Staubli VAL3: designr0.pjx

--- designr0.pjx ---
Parameters version=s7.6.2 stackSize=5000 millimeterUnit=true
Program file=start.pgx
Program file=stop.pgx
Data file=designr0.dtx

--- designr0.dtx ---
mdesc mNomSpeed
pointRx pikk[6 6]
  [0,0] = {x=-175.775864, y=339.495741, z=-126.071808, rx=0.004243, ry=-179.997236, rz=44.99886, fatherId=world[0]}
  [0,1] = {x=-182.38, y=339.495741, z=-126.071808, rx=0.004243, ry=-179.997236, rz=44.99886, fatherId=world[0]}
  [0,2] = {x=-188.98, y=339.5, z=-126, rx=180, ry=0, rz=-135, fatherId=world[0]}
  [0,3] = {x=-195.58, y=339.5, z=-126, rx=180, ry=0, rz=-135, fatherId=world[0]}
  [0,4] = {x=-202.18, y=339.5, z=-126, rx=180, ry=0, rz=-135, fatherId=world[0]}
  [0,5] = {x=-208.78, y=339.5, z=-126, rx=180, ry=0, rz=-135, fatherId=world[0]}
  [1,0] = {x=-175.78, y=349.8, z=-126, rx=180, ry=0, rz=-135, fatherId=world[0]}
  [1,1] = {x=-182.38, y=349.8, z=-126, rx=180, ry=0, rz=-135, fatherId=world[0]}
  [1,2] = {x=-188.98, y=349.8, z=-126, rx=180, ry=0, rz=-135, fatherId=world[0]}
  [1,3] = {x=-195.58, y=349.8, z=-126, rx=180, ry=0, rz=-135, fatherId=world[0]}
  [1,4] = {x=-202.18, y=349.8, z=-126, rx=180, ry=0, rz=-135, fatherId=world[0]}
  [1,5] = {x=-208.78, y=349.8, z=-126, rx=180, ry=0, rz=-135, fatherId=world[0]}
  [2,0] = {x=-175.78, y=360.1, z=-126, rx=180, ry=0, rz=-135, fatherId=world[0]}
  [2,1] = {x=-182.38, y=360.1, z=-126, rx=180, ry=0, rz=-135, fatherId=world[0]}
  [2,2] = {x=-188.98, y=360.1, z=-126, rx=180, ry=0, rz=-135, fatherId=world[0]}
  [2,3] = {x=-195.58, y=360.1, z=-126, rx=180, ry=0, rz=-135, fatherId=world[0]}
  [2,4] = {x=-202.18, y=360.1, z=-126, rx=180, ry=0, rz=-135, fatherId=world[0]}
  [2,5] = {x=-208.78, y=360.1, z=-126, rx=180, ry=0, rz=-135, fatherId=world[0]}
  [3,0] = {x=-175.78, y=370.4, z=-126, rx=180, ry=0, rz=-135, fatherId=world[0]}
  [3,1] = {x=-182.38, y=370.4, z=-126, rx=180, ry=0, rz=-135, fatherId=world[0]}
  [3,2] = {x=-188.98, y=370.4, z=-126, rx=180, ry=0, rz=-135, fatherId=world[0]}
  [3,3] = {x=-195.58, y=370.4, z=-126, rx=180, ry=0, rz=-135, fatherId=world[0]}
  [3,4] = {x=-202.18, y=370.4, z=-126, rx=180, ry=0, rz=-135, fatherId=world[0]}
  [3,5] = {x=-208.78, y=370.4, z=-126, rx=180, ry=0, rz=-135, fatherId=world[0]}
  [4,0] = {x=-175.78, y=380.7, z=-126, rx=180, ry=0, rz=-135, fatherId=world[0]}
  [4,1] = {x=-182.38, y=380.7, z=-126, rx=180, ry=0, rz=-135, fatherId=world[0]}
  [4,2] = {x=-188.98, y=380.7, z=-126, rx=180, ry=0, rz=-135, fatherId=world[0]}
  [4,3] = {x=-195.58, y=380.7, z=-126, rx=180, ry=0, rz=-135, fatherId=world[0]}
  [4,4] = {x=-202.18, y=380.7, z=-126, rx=180, ry=0, rz=-135, fatherId=world[0]}
  [4,5] = {x=-208.78, y=380.7, z=-126, rx=180, ry=0, rz=-135, fatherId=world[0]}
  [5,0] = {x=-175.78, y=391, z=-126, rx=180, ry=0, rz=-135, fatherId=world[0]}
  [5,1] = {x=-182.38, y=391, z=-126, rx=180, ry=0, rz=-135, fatherId=world[0]}
  [5,2] = {x=-188.98, y=391, z=-126, rx=180, ry=0, rz=-135, fatherId=world[0]}
  [5,3] = {x=-195.58, y=391, z=-126, rx=180, ry=0, rz=-135, fatherId=world[0]}
  [5,4] = {x=-202.18, y=391, z=-126, rx=180, ry=0, rz=-135, fatherId=world[0]}
  [5,5] = {x=-208.78, y=391, z=-126.071808, rx=0.004243, ry=-179.997236, rz=44.99886, fatherId=world[0]}
tool pick[6 6]
  [0,0] = {fatherId=flange[0], ioLink=valve1}
  [0,1] = {fatherId=flange[0], ioLink=valve1}
  [0,2] = {fatherId=flange[0], ioLink=valve1}
  [0,3] = {fatherId=flange[0], ioLink=valve1}
  [0,4] = {fatherId=flange[0], ioLink=valve1}
  [0,5] = {fatherId=flange[0], ioLink=valve1}
  [1,0] = {fatherId=flange[0], ioLink=valve1}
  [1,1] = {fatherId=flange[0], ioLink=valve1}
  [1,2] = {fatherId=flange[0], ioLink=valve1}
  [1,3] = {fatherId=flange[0], ioLink=valve1}
  [1,4] = {fatherId=flange[0], ioLink=valve1}
  [1,5] = {fatherId=flange[0], ioLink=valve1}
  [2,0] = {fatherId=flange[0], ioLink=valve1}
  [2,1] = {fatherId=flange[0], ioLink=valve1}
  [2,2] = {fatherId=flange[0], ioLink=valve1}
  [2,3] = {fatherId=flange[0], ioLink=valve1}
  [2,4] = {fatherId=flange[0], ioLink=valve1}
  [2,5] = {fatherId=flange[0], ioLink=valve1}
  [3,0] = {fatherId=flange[0], ioLink=valve1}
  [3,1] = {fatherId=flange[0], ioLink=valve1}
  [3,2] = {fatherId=flange[0], ioLink=valve1}
  [3,3] = {fatherId=flange[0], ioLink=valve1}
  [3,4] = {fatherId=flange[0], ioLink=valve1}
  [3,5] = {fatherId=flange[0], ioLink=valve1}
  [4,0] = {fatherId=flange[0], ioLink=valve1}
  [4,1] = {fatherId=flange[0], ioLink=valve1}
  [4,2] = {fatherId=flange[0], ioLink=valve1}
  [4,3] = {fatherId=flange[0], ioLink=valve1}
  [4,4] = {fatherId=flange[0], ioLink=valve1}
  [4,5] = {fatherId=flange[0], ioLink=valve1}
  [5,0] = {fatherId=flange[0], ioLink=valve1}
  [5,1] = {fatherId=flange[0], ioLink=valve1}
  [5,2] = {fatherId=flange[0], ioLink=valve1}
  [5,3] = {fatherId=flange[0], ioLink=valve1}
  [5,4] = {fatherId=flange[0], ioLink=valve1}
  [5,5] = {fatherId=flange[0], ioLink=valve1}
